FUNCTION Min3Value : lreal
VAR_INPUT
	a0:LREAL;
	a1:LREAL;
	a2:LREAL;
END_VAR
VAR
	b: LREAL;
END_VAR

b:=MIN(a0,a1);
IF b<a2 THEN
	 Min3Value:=b;
ELSE
	 Min3Value:=a2;
END_IF

END_FUNCTION

(* stored: Version 1.1.0.1, ProductVersion 3.1.4024.2
   POU Min3Value: Id {d3569c0e-c991-4a07-b224-6c72c55ebf19}, SpecialFunc None *)
